FUNCTION_BLOCK AX_TO_AR (* Composite FB for converting AX (BOOL) adapter to AR (REAL) adapter using F_SEL *)
  (* Standard: 61499-2; Description: Copyright (c) 2026 HR Agrartechnik GmbH This program and the accompanying materials are made available under the terms of the Eclipse Public License 2.0 which is available at https://www.eclipse.org/legal/epl-2.0/ SPDX-License-Identifier: EPL-2.0 *)
  (* Version 1.0, 2026-02-17, Franz Höpfinger, HR Agrartechnik GmbH *)
  PACKAGE adapter::conversion::unidirectional;
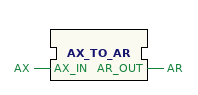
  SOCKETS
    AX_IN : adapter::types::unidirectional::AX; (* BOOL Adapter Input *)
  END_SOCKETS
  PLUGS
    AR_OUT : adapter::types::unidirectional::AR; (* REAL Adapter Output *)
  END_PLUGS
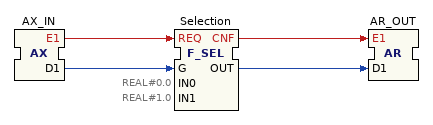
  FBS
    Selection : iec61131::selection::F_SEL(IN0 := REAL#0.0, IN1 := REAL#1.0);
  END_FBS
  EVENT_CONNECTIONS
    AX_IN.E1 TO Selection.REQ;
    Selection.CNF TO AR_OUT.E1;
  END_CONNECTIONS
  DATA_CONNECTIONS
    AX_IN.D1 TO Selection.G;
    Selection.OUT TO AR_OUT.D1;
  END_CONNECTIONS
END_FUNCTION_BLOCK
